TYPE ST_Color_Code :
STRUCT
	Pattern : UINT;
	Red :USINT;
	Green: USINT;
	Blue : USINT; 
END_STRUCT
END_TYPE

(* stored: Version 1.1.0.1, ProductVersion 3.1.4026.8
   DUT ST_Color_Code: Id {0ebbb323-0f58-4e03-9168-1c90dcb9dd81} *)
